// TIA Portal project "task2" (V16)
// Vorlageprojekt für das Buch mit Zielsystem S7-1200

(* hardware
DEVICE "S7-1200-Station_1"  S7-1200 Station
   slot 0: "Baugruppenträger_0"  Rack  V1.0
   slot 1: "PLC_1"  CPU 1211C DC/DC/DC  6ES7 211-1AE40-0XB0  V4.1
*)

// ===== PLC "PLC_1"  CPU 1211C DC/DC/DC =====

VAR_GLOBAL   // PLC tag table "Standard-Variablentabelle"
   "conv" AT %A0.0 : Bool;
   "start" AT %E0.0 : Bool;
   "stop" AT %E0.1 : Bool;
   "Tag_4" AT %I10.0 : Bool;
   "Tag_5" AT %Q10.0 : Bool;
   "Tag_6" AT %I10.1 : Bool;
   "x" AT %M0.0 : Bool;
   "Tag_1" AT %M0.1 : Bool;
   "diff1" AT %I0.7 : Bool;
   "Tag_2" AT %M0.3 : Bool;
   "diff2" AT %I1.0 : Bool;
   "pusher" AT %Q0.1 : Bool;
   "front" AT %I0.6 : Bool;
   "back" AT %I0.5 : Bool;
   "state1" AT %M1.0 : Bool;
   "stat1" AT %I0.2 : Bool;
   "state2" AT %M1.1 : Bool;
   "state2(1)" AT %I0.3 : Bool;
   "state0" AT %M1.2 : Bool;
   "Tag_3" AT %M2.2 : Bool;
   "Tag_7" AT %M3.0 : Bool;
   "Tag_8" AT %M5.1 : Bool;
   "Tag_9" AT %M5.3 : Bool;
   "Tag_10" AT %M4.4 : Bool;
   "Tag_11" AT %M4.5 : Bool;
END_VAR

// folder: System blocks/Program resources

DATA_BLOCK "t2"   // DB1
{ S7_Optimized_Access := 'TRUE' }
AUTHOR : Simatic
FAMILY : IEC
NAME : IEC_TMR
VERSION : 1.0
// stored: InstanceOfName IEC_TIMER
"IEC_TIMER"
BEGIN
END_DATA_BLOCK

// folder: (top level)

FUNCTION "MHJ-PLC-Lab-Function-S71200" : Void   // FC9000, SCL
{ S7_Optimized_Access := 'TRUE' }
VERSION : 0.1
   VAR_TEMP
      rdTimeReturn : Int;
      outputTime : DTL;
      SyncVal : Byte;
      forVal : Int;
      forVal_2 : Int;
      Value : Byte;
   END_VAR
   VAR CONSTANT
      CompVal : Byte := 16#34;
      Value_01 : Byte := 16#11;
      Value_01_DW : DWord := 16#A165_D992;
      Value_02_DW : DWord := 16#58BE_4401;
   END_VAR
BEGIN

   #Value:=PEEK(area := 16#82,
        dbNumber := 0,
        byteOffset := 511);
   #Value := #Value + 1;

   POKE(area := 16#82,
        dbNumber := 0,
        byteOffset := 511,
        value := #Value);

   POKE(area:=16#81,
        dbNumber:=0,
        byteOffset:=1016,
        value:=#Value_01_DW);
   POKE(area := 16#81,
        dbNumber := 0,
        byteOffset := 1020,
        value := #Value_02_DW);

   POKE(area := 16#81,
        dbNumber := 0,
        byteOffset := 511,
        value := B#16#00);

   FOR #forVal := 0 TO 120 DO
       FOR #forVal_2:=0 TO 10 DO
           #rdTimeReturn:=RD_SYS_T(#outputTime);
           #rdTimeReturn := WR_SYS_T(#outputTime);
           #rdTimeReturn := RD_SYS_T(#outputTime);
           #rdTimeReturn := WR_SYS_T(#outputTime);
       END_FOR;
       #SyncVal:= PEEK(area := 16#81,
                      dbNumber := 0,
                      byteOffset := 511);
       IF #SyncVal = #CompVal THEN
          GOTO M_1;
       END_IF;
   END_FOR;
   RETURN;

   M_1:
   POKE(area := 16#81,
        dbNumber := 0,
        byteOffset := 511,
        value := B#16#0);
END_FUNCTION

ORGANIZATION_BLOCK "Main"   // OB1, LAD, ProgramCycle
TITLE = "Main Program Sweep (Cycle)"
{ S7_Optimized_Access := 'TRUE' }
VERSION : 0.1
   VAR_INPUT
      Initial_Call : Bool;   // Initial call of this OB
      Remanence : Bool;   // =True, if remanent data are available
   END_VAR
   VAR_TEMP   // added for the SCL form of the ladder/FBD networks
      _w1 : Bool;
   END_VAR
BEGIN

REGION Network 1: Konnektierungsbaustein für PLC-Lab
   // Im Netzwerk 1 wird der Konnektierungsbaustein für PLC-Lab aufgerufen.
   // Dieser Aufruf darf nicht entfernt werden!
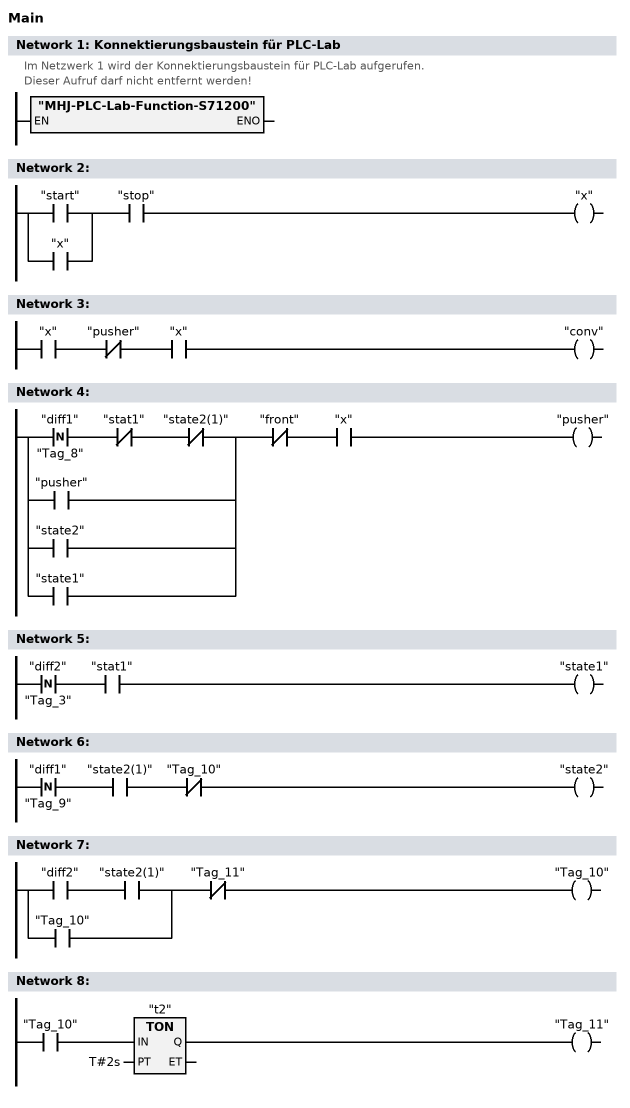
   RUNG wire#powerrail
      "MHJ-PLC-Lab-Function-S71200"()
   END_RUNG
   // the same network as SCL:
   "MHJ-PLC-Lab-Function-S71200"();
END_REGION

REGION Network 2
   RUNG wire#powerrail
      Contact( "start" )
      wire#w1
      Contact( "stop" )
      Coil( "x" )
   END_RUNG
   RUNG wire#powerrail
      Contact( "x" )
   END_RUNG wire#w1
   // the same network as SCL:
   "x" := ("start" OR "x") AND "stop";
END_REGION

REGION Network 3
   RUNG wire#powerrail
      Contact( "x" )
      I_Contact( "pusher" )
      Contact( "x" )
      Coil( "conv" )
   END_RUNG
   // the same network as SCL:
   "conv" := "x" AND NOT "pusher" AND "x";
END_REGION

REGION Network 4
   RUNG wire#powerrail
      N_Contact(operand := "diff1", bit := "Tag_8")
      I_Contact( "stat1" )
      I_Contact( "state2(1)" )
      wire#w1
      I_Contact( "front" )
      Contact( "x" )
      Coil( "pusher" )
   END_RUNG
   RUNG wire#powerrail
      Contact( "pusher" )
   END_RUNG wire#w1
   RUNG wire#powerrail
      Contact( "state2" )
   END_RUNG wire#w1
   RUNG wire#powerrail
      Contact( "state1" )
   END_RUNG wire#w1
   // the same network as SCL:
   #_w1 := NOT "diff1" AND "Tag_8";   // falling edge of "diff1"
   "Tag_8" := "diff1";
   "pusher" := ((#_w1 AND NOT "stat1" AND NOT "state2(1)") OR "pusher" OR "state2" OR "state1") AND NOT "front" AND "x";
END_REGION

REGION Network 5
   RUNG wire#powerrail
      N_Contact(operand := "diff2", bit := "Tag_3")
      Contact( "stat1" )
      Coil( "state1" )
   END_RUNG
   // the same network as SCL:
   #_w1 := NOT "diff2" AND "Tag_3";   // falling edge of "diff2"
   "Tag_3" := "diff2";
   "state1" := #_w1 AND "stat1";
END_REGION

REGION Network 6
   RUNG wire#powerrail
      N_Contact(operand := "diff1", bit := "Tag_9")
      Contact( "state2(1)" )
      I_Contact( "Tag_10" )
      Coil( "state2" )
   END_RUNG
   // the same network as SCL:
   #_w1 := NOT "diff1" AND "Tag_9";   // falling edge of "diff1"
   "Tag_9" := "diff1";
   "state2" := #_w1 AND "state2(1)" AND NOT "Tag_10";
END_REGION

REGION Network 7
   RUNG wire#powerrail
      Contact( "diff2" )
      Contact( "state2(1)" )
      wire#w1
      I_Contact( "Tag_11" )
      Coil( "Tag_10" )
   END_RUNG
   RUNG wire#powerrail
      Contact( "Tag_10" )
   END_RUNG wire#w1
   // the same network as SCL:
   "Tag_10" := (("diff2" AND "state2(1)") OR "Tag_10") AND NOT "Tag_11";
END_REGION

REGION Network 8
   "t2".TON(IN := "Tag_10", PT := T#2s);
   "Tag_11" := "t2".Q;
END_REGION
END_ORGANIZATION_BLOCK